// TIA Portal V20 export
DATA_BLOCK "BK24"   // DB271
// stored: MemoryReserve 100
   VAR
      "X10-1 SIDE TAPE ATTACHMENT #1 TOP VACUUM ON" : Bool;
      "X10-2 SIDE TAPE ATTACHMENT #1 TOP VACUUM OFF" : Bool;
      "X12-1 SIDE TAPE ATTACHMENT #1 BTM VACUUM ON" : Bool;
      "X12-2 SIDE TAPE ATTACHMENT #1 BTM VACUUM OFF" : Bool;
      "X14-1 SIDE TAPE ATTACHMENT #2 TOP VACUUM ON" : Bool;
      "X14-2 SIDE TAPE ATTACHMENT #2 TOP VACUUM OFF" : Bool;
      "X16-1 SIDE TAPE ATTACHMENT #2 BTM VACUUM ON" : Bool;
      "X16-2 SIDE TAPE ATTACHMENT #2 BTM VACUUM OFF" : Bool;
   END_VAR
BEGIN
END_DATA_BLOCK
